FUNCTION SPLIT_DWORD_INTO_BYTES (* this Function extracts the 4 BYTE from a dword *)
  (* Standard: 61499-1; Description: Copyright (c) 2025 HR Agrartechnik GmbH This program and the accompanying materials are made available under the terms of the Eclipse Public License 2.0 which is available at https://www.eclipse.org/legal/epl-2.0/ SPDX-License-Identifier: EPL-2.0 *)
  (* Version 1.0, 2025-12-21, Franz Höpfinger, HR Agrartechnik, initial Version *)
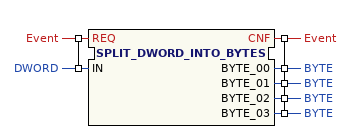
  EVENT_INPUT
    REQ WITH IN;
  END_EVENT
  EVENT_OUTPUT
    CNF WITH BYTE_00, BYTE_01, BYTE_02, BYTE_03;
  END_EVENT
  VAR_INPUT
    IN : DWORD;
  END_VAR
  VAR_OUTPUT
    BYTE_00 : BYTE;
    BYTE_01 : BYTE;
    BYTE_02 : BYTE;
    BYTE_03 : BYTE;
  END_VAR
  BODY IN ST:
(* this Function extracts the 4 BYTE from a dword *)
FUNCTION SPLIT_DWORD_INTO_BYTES

VAR_INPUT
	IN : DWORD;
END_VAR

VAR_OUTPUT
	BYTE_00 : BYTE;
	BYTE_01 : BYTE;
	BYTE_02 : BYTE;
	BYTE_03 : BYTE;
END_VAR

BYTE_00 := IN.%B0;
BYTE_01 := IN.%B1;
BYTE_02 := IN.%B2;
BYTE_03 := IN.%B3;

END_FUNCTION
  END_BODY
END_FUNCTION
